// TwinCAT 3 PLC project Hausaufgaben_FlipFlop
// ProgramVersion: 3.1.4026.16
// libraries:
//   Tc2_Standard, * (Beckhoff Automation GmbH)
//   Tc2_System, * (Beckhoff Automation GmbH)
// project tree:
//   / PlcTask.TcTTO
//   POUs/ FlipFlopR1.TcPOU, FlipFlopS1.TcPOU (not stored), MAIN.TcPOU (not stored), RSFlipFlop.TcPOU, ScaleFB.TcPOU, SRFlipFlop.TcPOU (not stored)
// real-time tasks:
//   TASK PlcTask: cycle T#10ms, priority 20, ADS port 350
//   TASK PlcTask1: cycle T#10ms, priority 21, ADS port 351
//   TASK PlcTask2: cycle T#10ms, priority 22, ADS port 352

CONFIGURATION Hausaufgaben_FlipFlop
    RESOURCE PLC ON TwinCAT3
        TASK PlcTask(INTERVAL := T#10ms, PRIORITY := 21);
        PROGRAM MAIN WITH PlcTask : MAIN;
    END_RESOURCE
END_CONFIGURATION

// ---- POUs/FlipFlopR1.TcPOU
FUNCTION_BLOCK FlipFlopR1 		//R-Dominanter FlipFlop
VAR_INPUT
	bSET: BOOL;					//Baustein-interne Set-Variable
	bRESET: BOOL;				//Baustein-interne Reset-Variable
END_VAR
VAR_OUTPUT
	bQ1: BOOL;					//Baustein-interne Ausgangs-Variable
END_VAR
VAR
END_VAR

IF bRESET 						//Abfrage ob Reset = 1, da R-Dominant
	THEN					
    bQ1 := FALSE;
ELSIF bSET AND NOT bRESET		//Abfrage ob Set = 1 und nicht Reset = 1
	THEN	
    bQ1 := TRUE;
END_IF;

END_FUNCTION_BLOCK

// ---- POUs/RSFlipFlop.TcPOU
FUNCTION_BLOCK RSFlipFlop
VAR_INPUT											//S-Dominanter RS-Baustein
	bSET: BOOL;										//Baustein-interne Set-Variable
	bRESET: BOOL;									//Baustein-interne Reset-Variable
END_VAR
VAR_OUTPUT
END_VAR
VAR
	RSFlipFlop: RS;									//Instanziierung des RS-Bausteins
END_VAR

RSFlipFlop(SET:= bSET, RESET1:= bRESET);			//Verknüpfung der Baustein-internen Variablen mit den Bausteineingängen

END_FUNCTION_BLOCK

// ---- POUs/ScaleFB.TcPOU
FUNCTION_BLOCK ScaleFB
VAR_INPUT
	iRohWert: INT;
END_VAR
VAR_OUTPUT
	ScaledValue: INT;
END_VAR
VAR
	NormMIN:INT:= 0;
	NormMAX:INT:= 27648;
	ScaleMIN:INT:= 0;
	ScaleMAX:INT:= 100;
END_VAR

ScaledValue:= ((ScaleMAX-ScaleMIN)*(iRohWert-NormMIN)/(NormMAX-NormMIN))+ScaleMIN;

END_FUNCTION_BLOCK
